// TIA Portal V20 export
DATA_BLOCK "SBK6"   // DB290
// stored: MemoryReserve 100
   VAR
      "X1-1 GATE EC SIDE TAPE PB.LOCK" : Bool;
      "X2-1 GATE EC SIDE TAPE PB.RESET" : Bool;
      "X3-1 SPARE" : Bool;
      "X4-1 SPARE" : Bool;
      "X1-2 GATE EC SIDE TAPE PB.UNLOCK" : Bool;
      "X2-2 SPARE" : Bool;
      "X3-2 SPARE" : Bool;
      "X4-2 SPARE" : Bool;
   END_VAR
BEGIN
END_DATA_BLOCK
